// SIMATIC S7-200 SMART project (STEP 7-Micro/WIN SMART), CPU SR40

ORGANIZATION_BLOCK 主程序:OB1
TITLE=程序注释
BEGIN
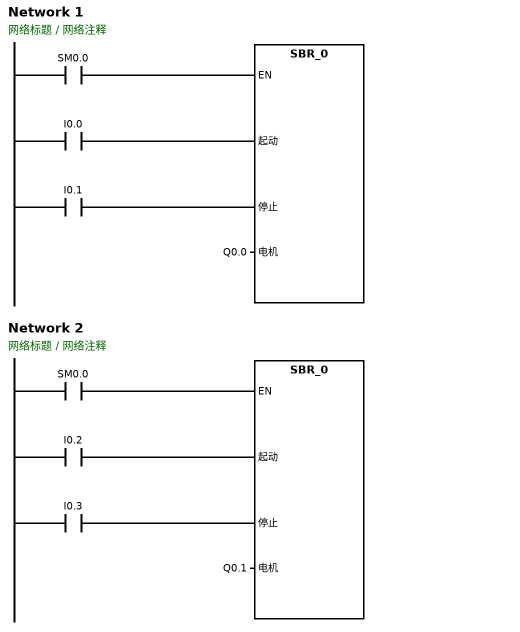
Network 1
// 网络标题
// 网络注释
// (network saved uncompiled; LAD cells follow)
// row 0: c0 -| |- SM0.0  c1 --  c2 [SBR_0 EN:=power@row0, 起动:=power@row1, 停止:=power@row2, 电机:=Q0.0]
// row 1: c0 -| |- I0.0  c1 --  c2 [box]
// row 2: c0 -| |- I0.1  c1 --  c2 [box]
// row 3: c2 [box]
Network 2
// 网络标题
// 网络注释
// (network saved uncompiled; LAD cells follow)
// row 0: c0 -| |- SM0.0  c1 --  c2 [SBR_0 EN:=power@row0, 起动:=power@row1, 停止:=power@row2, 电机:=Q0.1]
// row 1: c0 -| |- I0.2  c1 --  c2 [box]
// row 2: c0 -| |- I0.3  c1 --  c2 [box]
// row 3: c2 [box]
END_ORGANIZATION_BLOCK

SUBROUTINE_BLOCK SBR_0:SBR0
TITLE=子程序注释
VAR_INPUT
起动:BOOL;	// L0.0 
停止:BOOL;	// L0.1 
END_VAR
VAR_IN_OUT
电机:BOOL;	// L0.2 
END_VAR
BEGIN
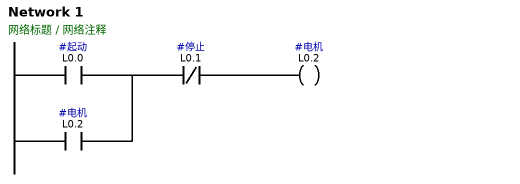
Network 1
// 网络标题
// 网络注释
LD     #起动:L0.0
O      #电机:L0.2
AN     #停止:L0.1
=      #电机:L0.2
END_SUBROUTINE_BLOCK
